# EPICS autosave request: ADAndorIstar/iocs/andorIstarIOC/iocBoot/iocAndorIstar/auto_settings.req
file "ADBase_settings.req",       P=$(P),  R=cam1:
#file "andorCCD_settings.req",     P=$(P),  R=cam1:
# Comment out the following line on Linux or if there is no Shamrock spectrograph on Windows
#file "shamrock_settings.req",     P=$(P),  R=sham1:
file "NDFile_settings.req",       P=$(P),  R=cam1:
file "NDPluginBase_settings.req", P=$(P),  R=image1:
file "NDStdArrays_settings.req",  P=$(P),  R=image1:
file "commonPlugin_settings.req", P=$(P)
